(*
SPDX-FileCopyrightText: © 2026 Oleksandr Tiutyk <trofimich@gmail.com>
SPDX-License-Identifier: MIT
License: https://opensource.org/license/mit
*)

(*!
<summary>Reports a field or property whose named type is not supported by the operation.</summary>
<description>
The caller identifies the unsupported member and type; this exception records their diagnostic description
rather than validating the member. Dynamic instances and clones belong to the current task memory manager
until cleanup. Dynamic copies are explicitly registered by Clone after construction; plain __NEW does not
transfer ownership to the task manager.
</description>
*)

{attribute 'enable_dynamic_creation'}
{attribute 'no_explicit_call' := 'do not call this function block directly'}
FUNCTION_BLOCK DataMemberTypeNotSupportedException EXTENDS GeneralException IMPLEMENTS IDataMemberTypeNotSupportedException
VAR_STAT
	//! <summary>Class name shared by all instances of this function block.</summary>
	{attribute 'hide'} 
	_ClassName : STRING := __POUNAME();
END_VAR

{attribute 'monitoring' := 'call'}
PROPERTY ClassName : REFERENCE TO STRING
GET
ClassName REF= _ClassName;
END_GET
END_PROPERTY

(*!
<summary>Creates a distinct DataMemberTypeNotSupportedException with copied diagnostics.</summary>
<description>
Preserves this concrete type and IDataMemberTypeNotSupportedException. Copies message, code, source and
timestamps through CopyGeneralFields; any prepared inner cause remains borrowed. The current task memory
manager owns the clone until cleanup. Allocation failure uses the shared terminal memory mechanism.
Descendants with additional payload must override Clone to preserve their type and fields. Registers the newly
constructed instance before copying payload, outside FB_init. Registration failure releases the unregistered
instance and raises a terminal error; copy failure leaves the registered instance owned by the task manager
for cleanup. Custom overrides must follow the same ownership sequence.
</description>
*)
METHOD Clone : IObject
VAR
	exceptionClone : POINTER TO DataMemberTypeNotSupportedException;
END_VAR
exceptionClone := __NEW(DataMemberTypeNotSupportedException);

IF exceptionClone = 0 THEN
	DynamicMemoryManager.RaiseAllocationFailure();
END_IF

DynamicMemoryManager.RegisterAutoDisposedObject(autoDisposedObject := exceptionClone^);

exceptionClone^.CopyGeneralFields(sourceException := THIS^);

Clone := exceptionClone^;
END_METHOD

(*!
<summary>Provides the library namespace used in diagnostics.</summary>
<description>
Borrowed read-only reference to the compiler-initialized library namespace; no ownership transfer.
</description>
*)
{attribute 'monitoring' := 'call'}
PROPERTY NamespaceName : REFERENCE TO STRING
GET
NamespaceName REF= CurrentNamespace.Name;
END_GET
END_PROPERTY

(*!
<summary>Reports the byte size of this concrete instance.</summary>
<description>
Uses XSIZEOF on the instance. Does not include separately allocated payloads or prove that an arbitrary
address is valid.
</description>
*)
{attribute 'monitoring' := 'call'}
PROPERTY SelfSize : ULINT
GET
SelfSize := XSIZEOF(THIS^);
END_GET
END_PROPERTY

(*!
<summary>Formats the rejected member and propagates the exception.</summary>
<description>
Call in the owning cyclic task, not during FB_init. Builds a member diagnostic without heap allocation during
message preparation and captures source and timestamps with zero error code and no inner cause. Input storage
is not retained. Exception clone allocation failure uses the shared terminal memory mechanism.
</description>
<param name="dataMemberName">Name of the field or property rejected by the caller.</param>
<param name="dataMemberTypeName">Name of the unsupported concrete type.</param>
*)
METHOD Throw
VAR_INPUT
	sourceNamespaceName : STRING;
	sourceClassName : STRING;
	sourcePOUName : STRING;
	sourcePosition : STRING;
	dataMemberName : STRING;
	dataMemberTypeName : STRING;
END_VAR
VAR
	message : ERROR_MESSAGE;
END_VAR
WideStrings.Append255(
	message,
	"Field or property '",
	TO_WSTRING(dataMemberName),
	"' has not supported type '",
	TO_WSTRING(dataMemberTypeName),
	"' in the instance of '",
	TO_WSTRING(sourceNamespaceName),
	".",
	TO_WSTRING(sourceClassName),
	"'");

InternalThrow(
	sourceNamespaceName := sourceNamespaceName,
	sourceClassName := sourceClassName,
	sourcePOUName := sourcePOUName,
	sourcePosition := sourcePosition,
	message := message,
	errorCode := 0,
	innerException := 0
);
END_METHOD

END_FUNCTION_BLOCK

(* stored: Version 1.1.0.1
   POU DataMemberTypeNotSupportedException: Id {9e878d14-6b39-4fa7-a91f-ceec4cab8cd2}, SpecialFunc None
   Property ClassName: Id {f8773de5-989e-46ed-bd87-50902874630e}
   Get Get: Id {377bd033-1bd8-44bb-b9de-80387fff9780}
   Method Clone: Id {9b92cfed-830e-491f-8f68-5b6ad0ab5a78}
   Property NamespaceName: Id {0352b25f-d4f2-402a-a14d-e0520aa97aa7}
   Get Get: Id {b87faf39-8de2-43c7-85ee-e47b96fd4417}
   Property SelfSize: Id {3d0eb1ca-033b-41be-9e09-02fc5254f11d}
   Get Get: Id {62217dcd-f83a-48cf-9bc3-a0703d997c98}
   Method Throw: Id {7ca82ec6-4830-4a12-b105-1131d118f378} *)
